TYPE ST_SolenoidSet :
STRUCT
	
	bSolenoidA 		: BOOL;  // Válvula Solenoide A 
    bSolenoidB 		: BOOL;  // Válvula Solenoide B 
    bSolenoidC 		: BOOL;  // Válvula Solenoide C 
	
END_STRUCT
END_TYPE

(* stored: Version 1.1.0.1, ProductVersion 3.1.4024.15
   DUT ST_SolenoidSet: Id {c0450522-fb26-4722-8a4c-9b7935364899} *)
